// TIA Portal V17 export
// export: Created 2022-03-12T16:05:34.6811471Z, ExportSetting WithDefaults, DisplayName Totally Integrated Automation Portal, DisplayVersion V17, DisplayName TIA Portal Openness, DisplayVersion V17, DisplayName TIA Portal Version Control Interface, DisplayVersion V17, DisplayName STEP 7 Professional, DisplayVersion V17, DisplayName STEP 7 Safety, DisplayVersion V17, DisplayName WinCC Advanced / Unified PC, DisplayVersion V17
TYPE "CPG_typeSortFilter"
// stored: IsFailsafeCompliant false
   STRUCT
      cmdFilterActiveEvents : Bool;   // Filter for Active events: 1=only show active events; 0=show all events
      cmdFilterCategory : Bool;   // Filter by Category: filter events to show only selected category number
      cmdSortCategory : Bool;   // Sort by Category: 1=sort events by ascending category number
      cfgTimeSortDirection : Bool;   // Sort by Time: 1=newest first; 0=oldest first
      cfgEventListOffset : Int;   // Commanded event list offset (used for scrolling)
      cfgFilterCategory : Int;   // Filter by Category: filtered category number
   END_STRUCT;
END_TYPE
